// TIA Portal V18 export
// export: Created 2026-06-23T08:49:29.7033678Z, ExportSetting WithDefaults, DisplayName Totally Integrated Automation Portal, DisplayVersion V18, DisplayName TIA Portal Openness, DisplayVersion V18, DisplayName TIA Portal Version Control Interface, DisplayVersion V18, DisplayName STEP 7 Professional, DisplayVersion V18, DisplayName STEP 7 Safety, DisplayVersion V18, DisplayName WinCC Professional, DisplayVersion V18
FUNCTION "FC_HMI_Animation_PLC1" : Void   // FC60, LAD
{ S7_Optimized_Access := 'TRUE' }
VERSION : 0.1
// stored: AutoNumber true, IsIECCheckEnabled false, SetENOAutomatically false, UDAEnableTagReadback false
BEGIN

REGION Network 1: Cánh khuấy Bồn 1: Tăng khung hình khi chạy
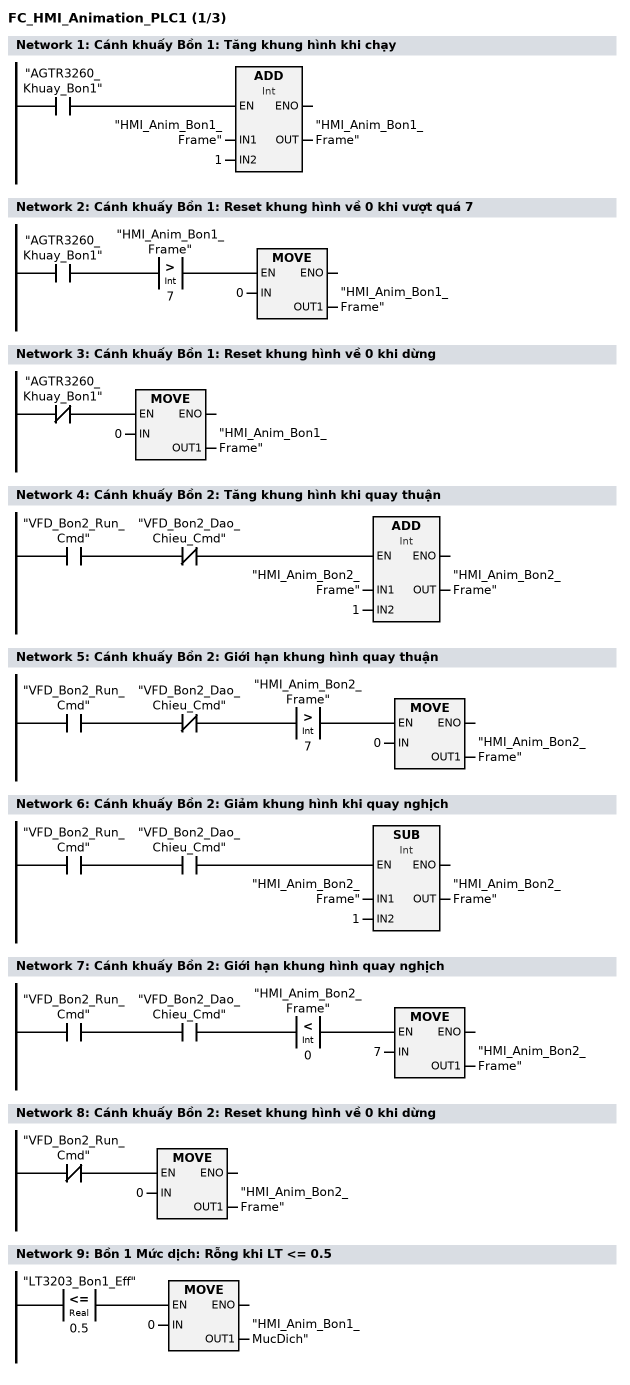
   RUNG wire#powerrail
      Contact( "AGTR3260_Khuay_Bon1" )
      { S7_Templates := "SrcType := Int"; S7_GenerateENO := "TRUE" } Add(in1 := "HMI_Anim_Bon1_Frame", in2 := 1, out => "HMI_Anim_Bon1_Frame")
   END_RUNG
   // the same network as SCL:
   IF "AGTR3260_Khuay_Bon1" THEN "HMI_Anim_Bon1_Frame" := "HMI_Anim_Bon1_Frame" + 1; END_IF;
END_REGION

REGION Network 2: Cánh khuấy Bồn 1: Reset khung hình về 0 khi vượt quá 7
   RUNG wire#powerrail
      Contact( "AGTR3260_Khuay_Bon1" )
      { S7_Templates := "SrcType := Int" } GT_Contact(in1 := "HMI_Anim_Bon1_Frame", in2 := 7)
      { S7_GenerateENO := "TRUE" } Move(in := 0, out1 => "HMI_Anim_Bon1_Frame")
   END_RUNG
   // the same network as SCL:
   IF "AGTR3260_Khuay_Bon1" AND ("HMI_Anim_Bon1_Frame" > 7) THEN "HMI_Anim_Bon1_Frame" := 0; END_IF;
END_REGION

REGION Network 3: Cánh khuấy Bồn 1: Reset khung hình về 0 khi dừng
   RUNG wire#powerrail
      I_Contact( "AGTR3260_Khuay_Bon1" )
      { S7_GenerateENO := "TRUE" } Move(in := 0, out1 => "HMI_Anim_Bon1_Frame")
   END_RUNG
   // the same network as SCL:
   IF NOT "AGTR3260_Khuay_Bon1" THEN "HMI_Anim_Bon1_Frame" := 0; END_IF;
END_REGION

REGION Network 4: Cánh khuấy Bồn 2: Tăng khung hình khi quay thuận
   RUNG wire#powerrail
      Contact( "VFD_Bon2_Run_Cmd" )
      I_Contact( "VFD_Bon2_Dao_Chieu_Cmd" )
      { S7_Templates := "SrcType := Int"; S7_GenerateENO := "TRUE" } Add(in1 := "HMI_Anim_Bon2_Frame", in2 := 1, out => "HMI_Anim_Bon2_Frame")
   END_RUNG
   // the same network as SCL:
   IF "VFD_Bon2_Run_Cmd" AND NOT "VFD_Bon2_Dao_Chieu_Cmd" THEN
       "HMI_Anim_Bon2_Frame" := "HMI_Anim_Bon2_Frame" + 1;
   END_IF;
END_REGION

REGION Network 5: Cánh khuấy Bồn 2: Giới hạn khung hình quay thuận
   RUNG wire#powerrail
      Contact( "VFD_Bon2_Run_Cmd" )
      I_Contact( "VFD_Bon2_Dao_Chieu_Cmd" )
      { S7_Templates := "SrcType := Int" } GT_Contact(in1 := "HMI_Anim_Bon2_Frame", in2 := 7)
      { S7_GenerateENO := "TRUE" } Move(in := 0, out1 => "HMI_Anim_Bon2_Frame")
   END_RUNG
   // the same network as SCL:
   IF "VFD_Bon2_Run_Cmd" AND NOT "VFD_Bon2_Dao_Chieu_Cmd" AND ("HMI_Anim_Bon2_Frame" > 7) THEN
       "HMI_Anim_Bon2_Frame" := 0;
   END_IF;
END_REGION

REGION Network 6: Cánh khuấy Bồn 2: Giảm khung hình khi quay nghịch
   RUNG wire#powerrail
      Contact( "VFD_Bon2_Run_Cmd" )
      Contact( "VFD_Bon2_Dao_Chieu_Cmd" )
      { S7_Templates := "SrcType := Int"; S7_GenerateENO := "TRUE" } Sub(in1 := "HMI_Anim_Bon2_Frame", in2 := 1, out => "HMI_Anim_Bon2_Frame")
   END_RUNG
   // the same network as SCL:
   IF "VFD_Bon2_Run_Cmd" AND "VFD_Bon2_Dao_Chieu_Cmd" THEN
       "HMI_Anim_Bon2_Frame" := "HMI_Anim_Bon2_Frame" - 1;
   END_IF;
END_REGION

REGION Network 7: Cánh khuấy Bồn 2: Giới hạn khung hình quay nghịch
   RUNG wire#powerrail
      Contact( "VFD_Bon2_Run_Cmd" )
      Contact( "VFD_Bon2_Dao_Chieu_Cmd" )
      { S7_Templates := "SrcType := Int" } LT_Contact(in1 := "HMI_Anim_Bon2_Frame", in2 := 0)
      { S7_GenerateENO := "TRUE" } Move(in := 7, out1 => "HMI_Anim_Bon2_Frame")
   END_RUNG
   // the same network as SCL:
   IF "VFD_Bon2_Run_Cmd" AND "VFD_Bon2_Dao_Chieu_Cmd" AND ("HMI_Anim_Bon2_Frame" < 0) THEN
       "HMI_Anim_Bon2_Frame" := 7;
   END_IF;
END_REGION

REGION Network 8: Cánh khuấy Bồn 2: Reset khung hình về 0 khi dừng
   RUNG wire#powerrail
      I_Contact( "VFD_Bon2_Run_Cmd" )
      { S7_GenerateENO := "TRUE" } Move(in := 0, out1 => "HMI_Anim_Bon2_Frame")
   END_RUNG
   // the same network as SCL:
   IF NOT "VFD_Bon2_Run_Cmd" THEN "HMI_Anim_Bon2_Frame" := 0; END_IF;
END_REGION

REGION Network 9: Bồn 1 Mức dịch: Rỗng khi LT <= 0.5
   RUNG wire#powerrail
      { S7_Templates := "SrcType := Real" } LE_Contact(in1 := "LT3203_Bon1_Eff", in2 := 0.5)
      { S7_GenerateENO := "TRUE" } Move(in := 0, out1 => "HMI_Anim_Bon1_MucDich")
   END_RUNG
   // the same network as SCL:
   IF "LT3203_Bon1_Eff" <= 0.5 THEN "HMI_Anim_Bon1_MucDich" := 0; END_IF;
END_REGION

REGION Network 10: Bồn 1 Mức dịch: Mức 40% khi 0.5 < LT < 50.0
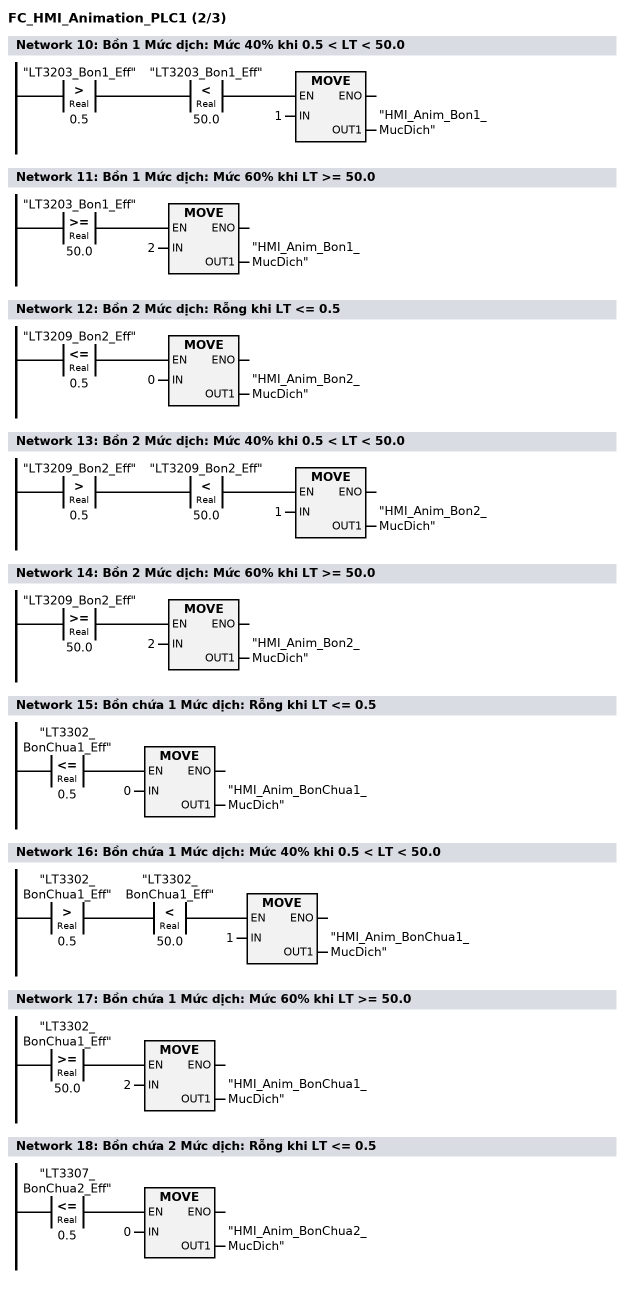
   RUNG wire#powerrail
      { S7_Templates := "SrcType := Real" } GT_Contact(in1 := "LT3203_Bon1_Eff", in2 := 0.5)
      { S7_Templates := "SrcType := Real" } LT_Contact(in1 := "LT3203_Bon1_Eff", in2 := 50.0)
      { S7_GenerateENO := "TRUE" } Move(in := 1, out1 => "HMI_Anim_Bon1_MucDich")
   END_RUNG
   // the same network as SCL:
   IF ("LT3203_Bon1_Eff" > 0.5) AND ("LT3203_Bon1_Eff" < 50.0) THEN "HMI_Anim_Bon1_MucDich" := 1; END_IF;
END_REGION

REGION Network 11: Bồn 1 Mức dịch: Mức 60% khi LT >= 50.0
   RUNG wire#powerrail
      { S7_Templates := "SrcType := Real" } GE_Contact(in1 := "LT3203_Bon1_Eff", in2 := 50.0)
      { S7_GenerateENO := "TRUE" } Move(in := 2, out1 => "HMI_Anim_Bon1_MucDich")
   END_RUNG
   // the same network as SCL:
   IF "LT3203_Bon1_Eff" >= 50.0 THEN "HMI_Anim_Bon1_MucDich" := 2; END_IF;
END_REGION

REGION Network 12: Bồn 2 Mức dịch: Rỗng khi LT <= 0.5
   RUNG wire#powerrail
      { S7_Templates := "SrcType := Real" } LE_Contact(in1 := "LT3209_Bon2_Eff", in2 := 0.5)
      { S7_GenerateENO := "TRUE" } Move(in := 0, out1 => "HMI_Anim_Bon2_MucDich")
   END_RUNG
   // the same network as SCL:
   IF "LT3209_Bon2_Eff" <= 0.5 THEN "HMI_Anim_Bon2_MucDich" := 0; END_IF;
END_REGION

REGION Network 13: Bồn 2 Mức dịch: Mức 40% khi 0.5 < LT < 50.0
   RUNG wire#powerrail
      { S7_Templates := "SrcType := Real" } GT_Contact(in1 := "LT3209_Bon2_Eff", in2 := 0.5)
      { S7_Templates := "SrcType := Real" } LT_Contact(in1 := "LT3209_Bon2_Eff", in2 := 50.0)
      { S7_GenerateENO := "TRUE" } Move(in := 1, out1 => "HMI_Anim_Bon2_MucDich")
   END_RUNG
   // the same network as SCL:
   IF ("LT3209_Bon2_Eff" > 0.5) AND ("LT3209_Bon2_Eff" < 50.0) THEN "HMI_Anim_Bon2_MucDich" := 1; END_IF;
END_REGION

REGION Network 14: Bồn 2 Mức dịch: Mức 60% khi LT >= 50.0
   RUNG wire#powerrail
      { S7_Templates := "SrcType := Real" } GE_Contact(in1 := "LT3209_Bon2_Eff", in2 := 50.0)
      { S7_GenerateENO := "TRUE" } Move(in := 2, out1 => "HMI_Anim_Bon2_MucDich")
   END_RUNG
   // the same network as SCL:
   IF "LT3209_Bon2_Eff" >= 50.0 THEN "HMI_Anim_Bon2_MucDich" := 2; END_IF;
END_REGION

REGION Network 15: Bồn chứa 1 Mức dịch: Rỗng khi LT <= 0.5
   RUNG wire#powerrail
      { S7_Templates := "SrcType := Real" } LE_Contact(in1 := "LT3302_BonChua1_Eff", in2 := 0.5)
      { S7_GenerateENO := "TRUE" } Move(in := 0, out1 => "HMI_Anim_BonChua1_MucDich")
   END_RUNG
   // the same network as SCL:
   IF "LT3302_BonChua1_Eff" <= 0.5 THEN "HMI_Anim_BonChua1_MucDich" := 0; END_IF;
END_REGION

REGION Network 16: Bồn chứa 1 Mức dịch: Mức 40% khi 0.5 < LT < 50.0
   RUNG wire#powerrail
      { S7_Templates := "SrcType := Real" } GT_Contact(in1 := "LT3302_BonChua1_Eff", in2 := 0.5)
      { S7_Templates := "SrcType := Real" } LT_Contact(in1 := "LT3302_BonChua1_Eff", in2 := 50.0)
      { S7_GenerateENO := "TRUE" } Move(in := 1, out1 => "HMI_Anim_BonChua1_MucDich")
   END_RUNG
   // the same network as SCL:
   IF ("LT3302_BonChua1_Eff" > 0.5) AND ("LT3302_BonChua1_Eff" < 50.0) THEN
       "HMI_Anim_BonChua1_MucDich" := 1;
   END_IF;
END_REGION

REGION Network 17: Bồn chứa 1 Mức dịch: Mức 60% khi LT >= 50.0
   RUNG wire#powerrail
      { S7_Templates := "SrcType := Real" } GE_Contact(in1 := "LT3302_BonChua1_Eff", in2 := 50.0)
      { S7_GenerateENO := "TRUE" } Move(in := 2, out1 => "HMI_Anim_BonChua1_MucDich")
   END_RUNG
   // the same network as SCL:
   IF "LT3302_BonChua1_Eff" >= 50.0 THEN "HMI_Anim_BonChua1_MucDich" := 2; END_IF;
END_REGION

REGION Network 18: Bồn chứa 2 Mức dịch: Rỗng khi LT <= 0.5
   RUNG wire#powerrail
      { S7_Templates := "SrcType := Real" } LE_Contact(in1 := "LT3307_BonChua2_Eff", in2 := 0.5)
      { S7_GenerateENO := "TRUE" } Move(in := 0, out1 => "HMI_Anim_BonChua2_MucDich")
   END_RUNG
   // the same network as SCL:
   IF "LT3307_BonChua2_Eff" <= 0.5 THEN "HMI_Anim_BonChua2_MucDich" := 0; END_IF;
END_REGION

REGION Network 19: Bồn chứa 2 Mức dịch: Mức 40% khi 0.5 < LT < 50.0
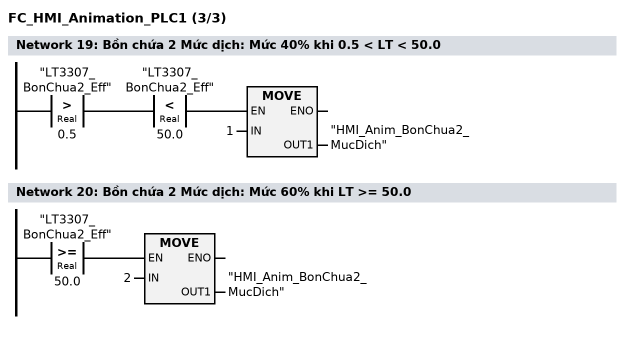
   RUNG wire#powerrail
      { S7_Templates := "SrcType := Real" } GT_Contact(in1 := "LT3307_BonChua2_Eff", in2 := 0.5)
      { S7_Templates := "SrcType := Real" } LT_Contact(in1 := "LT3307_BonChua2_Eff", in2 := 50.0)
      { S7_GenerateENO := "TRUE" } Move(in := 1, out1 => "HMI_Anim_BonChua2_MucDich")
   END_RUNG
   // the same network as SCL:
   IF ("LT3307_BonChua2_Eff" > 0.5) AND ("LT3307_BonChua2_Eff" < 50.0) THEN
       "HMI_Anim_BonChua2_MucDich" := 1;
   END_IF;
END_REGION

REGION Network 20: Bồn chứa 2 Mức dịch: Mức 60% khi LT >= 50.0
   RUNG wire#powerrail
      { S7_Templates := "SrcType := Real" } GE_Contact(in1 := "LT3307_BonChua2_Eff", in2 := 50.0)
      { S7_GenerateENO := "TRUE" } Move(in := 2, out1 => "HMI_Anim_BonChua2_MucDich")
   END_RUNG
   // the same network as SCL:
   IF "LT3307_BonChua2_Eff" >= 50.0 THEN "HMI_Anim_BonChua2_MucDich" := 2; END_IF;
END_REGION
END_FUNCTION
